FUNCTION_BLOCK HaltTask EXTENDS TcoCore.TcoTask IMPLEMENTS ITcoDriveSimple
VAR
    {attribute addProperty Name "<#Deceleration#>"}
    _deceleration : LREAL;
    {attribute addProperty Name "<#Jerk#>"}
    _jerk : LREAL;
END_VAR
VAR
    {attribute 'hide'}
    _axisRef : REFERENCE TO TcoAxisRef;
    {attribute 'hide'}
    _mcHalt : Tc2_MC2.MC_Halt;
END_VAR

IF NOT __ISVALIDREF(_axisRef) THEN
    IF __ISVALIDREF(DriveRef) THEN
        _axisRef REF= DriveRef.AxisRef;
    ELSE
        RETURN;
    END_IF
END_IF

IF Execute() THEN
    _mcHalt(Axis := _axisRef);

    IF _mcHalt.CommandAborted THEN
        THIS^.Abort();
    END_IF

    DoneWhen(_mcHalt.Done);
    ThrowWhen(_mcHalt.Error);
END_IF

PROPERTY DriveRef : REFERENCE TO TcoDriveSimple
GET
VAR
    _drive : ITcoDriveSimple := 0;
END_VAR
IF __QUERYINTERFACE(THIS^._Parent, _drive) THEN
    DriveRef REF= _drive.DriveRef;
END_IF
END_GET
END_PROPERTY

METHOD PUBLIC FB_init : BOOL
VAR_INPUT
    bInitRetains : BOOL; // if TRUE, the retain variables are initialized (warm start / cold start)
    bInCopyCode : BOOL; // if TRUE, the instance afterwards gets moved into the copy code (online change)
    Parent : ITcoObject;
END_VAR
SUPER^.FB_init(bInitRetains := bInitRetains, bInCopyCode := bInCopyCode, Parent := Parent);
END_METHOD

METHOD INTERNAL InvokeWithParams : ITcoTaskStatus
VAR_INPUT
    inDeceleration : LREAL;
    inJerk : LREAL;
END_VAR
_deceleration := inDeceleration;
_jerk := inJerk;
InvokeWithParams := THIS^.Invoke();
END_METHOD

(*~
	<docu>
		<summary>
			Executes when task is aborted.
		</summary>			
	</docu>	
~*)
METHOD PROTECTED OnAbort
_mcHalt(Axis := _axisRef, Execute := FALSE, Deceleration := _deceleration);
THIS^.DriveRef._movementState.Restore();
END_METHOD

(*~
	<docu>
		<summary>
			Executes when task reaches the ```Done``` state .
		</summary>			
	</docu>	
~*)
METHOD PROTECTED OnDone
_mcHalt(Axis := _axisRef, Execute := FALSE, Deceleration := _deceleration);
THIS^.DriveRef._movementState.Restore();
END_METHOD

(*~
	<docu>
		<summary>
			Executes when task reaches the ```Error``` state.
			<para>
				Do not confuse with <see cref="TcoTask.PlcTcoTask.WhileError()"/>, that is called cyclically until '''Error''' state is left.
			</para>
		</summary>			
	</docu>	
~*)
METHOD PROTECTED OnError
THIS^.DriveRef._movementState.Restore();

IF NOT _axisRef.Status.Error THEN
	DriveRef.SetErrorID(DriveRef._haltTask._mcHalt.ErrorID);
END_IF
_mcHalt(Axis := _axisRef, Execute := FALSE);
END_METHOD

METHOD PROTECTED OnStart
_mcHalt(Axis := _axisRef, Execute := false, Deceleration := _deceleration);
_mcHalt(Axis := _axisRef, Execute := TRUE, Deceleration := _deceleration);
END_METHOD

(*~
	<docu>
		<summary>
			Restores this instance to the Ready state. Can be called explicitly or from within one of the restore mechanisms.
			<para>
				See also <see cref="TcoTask.PlcTcoTask.AutoRestorable()"/>
			</para>
		</summary>			
	</docu>	
~*)
METHOD Restore : ITcoRestorable
SUPER^.Restore();
END_METHOD

(*~
	<docu>
		<summary>
			Executes until task is in ```Error``` state .
		</summary>			
	</docu>	
~*)
METHOD PROTECTED WhileError
IF NOT _axisRef.Status.Error THEN
	DriveRef.SetErrorID(DriveRef._haltTask._mcHalt.ErrorID);
    _mcHalt(Axis := _axisRef, Execute := FALSE);
END_IF
END_METHOD

END_FUNCTION_BLOCK

(* stored: Version 1.1.0.1, ProductVersion 3.1.4024.9
   POU HaltTask: Id {7b2095f5-1f56-0a11-251d-e8dd47e39c60}, SpecialFunc None
   Property DriveRef: Id {05a8f2c1-5c4a-032e-391c-6015609bba63}
   Get Get: Id {c577432b-6bf0-02c1-2d8c-999bc8637657}
   Method FB_init: Id {d2ee9d25-2557-0248-1e0b-2092fdeb9e20}
   Method InvokeWithParams: Id {e0f5b9d1-b2ab-028e-0981-014cb0964a83}
   Method OnAbort: Id {9cde54a8-1b2e-0c32-0afa-bf3ad991b9e0}
   Method OnDone: Id {28ff8f2d-bf50-0b5a-1ad1-14f70e4986bb}
   Method OnError: Id {2aa19486-3273-0dcb-3fca-71dc00c2ea0a}
   Method OnStart: Id {7c680306-98e9-0c27-1b7f-0179e6eebe7c}
   Method Restore: Id {5b189d9a-d345-0f25-1831-45a12b9aee90}
   Method WhileError: Id {18785d6e-b3bd-04ec-1a40-8d17a3911928} *)
